{attribute 'qualified_only'}
VAR_GLOBAL
	startButton : button;
	stopButton : button;
	start_Button : BOOL;
	stop_Button : BOOL;
	mode_button : enum_switch := 0;
	rotSwitch : BOOL;
	vir_man_indi : vir_man_status;
END_VAR

(* stored: Version 1.1.0.1, ProductVersion 3.1.4024.12
   GVL GVL: Id {b0ccc028-8130-4d40-ace7-24fcdb9805e2} *)
